{attribute 'linkalways'} 
{attribute 'no_explicit_call' := 'This FB is a CLASS and must be accessed using methods or properties'}
{attribute 'enable_dynamic_creation'}
FUNCTION_BLOCK Node_F_VN_OCR EXTENDS VisionNode
VAR
	ipSrcImage : _ITcVnImage;
    eModel : _ETcVnOcrModelType(ETcVnOcrModelType.TCVN_OMT_NUMBERS);
    ipCharacters : _ITcVnContainer;
    hrPrev : _HRESULT(S_OK);
	hresult : _HRESULT(S_OK);
END_VAR

//TODO This function requires the use of FB_InitializeFunction function block.

METHOD PUBLIC  Clone : I_Node
VAR
	pNode : POINTER TO Node_F_VN_OCR;
END_VAR
pNode := __NEW(Node_F_VN_OCR);
Clone := pNode^;
END_METHOD

METHOD FB_init : BOOL
VAR_INPUT
	bInitRetains : BOOL; // if TRUE, the retain variables are initialized (warm start / cold start)
	bInCopyCode : BOOL;  // if TRUE, the instance afterwards gets moved into the copy code (online change)
END_VAR
AddInput('ipSrcImage', ipSrcImage);
AddParameter('eModel', eModel);
AddInput('hrPrev', hrPrev);
AddOutput('ipCharacters', ipCharacters);
AddOutput('hresult',hresult);
END_METHOD

METHOD PROTECTED OnExecute
hresult.Value := F_VN_OCR(
	ipSrcImage := ipSrcImage.Value,
    eModel := eModel.Value,
	ipCharacters := ipCharacters.Value,
	hrPrev:= hrPrev.Value);
END_METHOD

METHOD PUBLIC PreExecutionCheck
VAR_INPUT
	Check : I_PreExecutionChecks;
END_VAR
Check.IsTrue(ipSrcImage.IsValid, 'ipSrcImage must contain an image');
Check.IsTrue(ipSrcImage.IsPixelDepth(8), 'ipSrcImage must have 8 bit pixel depth');
Check.IsTrue(ipSrcImage.HasChannelCount(1), 'ipSrcImage must contain 1 channel');
END_METHOD

END_FUNCTION_BLOCK

(* stored: Version 1.1.0.1, ProductVersion 3.1.4024.13
   POU Node_F_VN_OCR: Id {0af6b6c4-6110-00fa-2380-c1a161cf2841}, SpecialFunc None
   Folder Constructor: Id {3d8e3bfd-03a2-08d1-1cca-49c5a2886041}
   Method Clone: Id {be79d7ce-06e2-0331-0b24-9a394559f903}
   Method FB_init: Id {18da78b1-fe20-06ae-28da-5505362f439b}
   Method OnExecute: Id {5f2ff8d6-c3ce-02bd-0489-8b1e62c2629c}
   Method PreExecutionCheck: Id {ce43c0eb-49b7-0d5e-259f-e72138b3455f} *)
